TEXTLIST TaskText
  0 = 'No Text'
  1 = 'Not Started'
  2 = 'Started'
  3 = 'Completed'
  4 = 'Passed'
  5 = 'Failed'
  6 = 'Rejected'
  7 = 'Skipped'
  8 = 'Bypassed'
  9 = 'Unknown'
   = ''
END_TEXTLIST

(* stored: Version 1.1.0.1, ProductVersion 3.1.4024.12
   TextList TaskText: Id {4b70b591-efbf-4a9b-9cb3-5a346e79b143} *)
